// TIA Portal V18 export
DATA_BLOCK "FB21-Flush A_DB_1"   // DB160
VERSION : 0.1
// stored: AutoNumber true, DBAccessibleFromOPCUA true, InstanceOfName FB21-Flush A, InstanceOfType FB
"FB21-Flush A"
   // VAR_INPUT
   //    "Time" : DInt;
   //    "Pump ON delay" : DInt;
   //    "Pump OFF delay" : DInt;
   // END_VAR
   // VAR_OUTPUT
   //    "dispensing Time PV" : Int;
   // END_VAR
   // VAR_IN_OUT
   //    start : Bool;
   //    "Stop Flush" : Bool;
   //    "Flush  Running" : Bool;
   //    "Flush completed" : Bool;
   //    "ON Gear Pump" : Bool;
   // END_VAR
   // VAR
   //    "dispensing time done" : Bool;
   //    "dispensing time in sec" : DInt;
   //    "timer input" : DInt;
   //    IEC_Timer_0_Instance { S7_SetPoint := 'True'} : TON_TIME;
   //    IEC_Timer_0_Instance_1 { S7_SetPoint := 'True'} : TON_TIME;
   //    IEC_Timer_0_Instance_2 { S7_SetPoint := 'True'} : TON_TIME;
   //    IEC_Timer_0_Instance_3 { S7_SetPoint := 'True'} : TON_TIME;
   // END_VAR
BEGIN
END_DATA_BLOCK
